# B&R Automation Studio project MotionTestBenchMaster (part 52)

```iecst
                               VAR_DOS_SEQ.Device.LSJ200.ALR := FALSE;                                                 (* STEP: 67 *)
                               VAR_DOS_SEQ.Device.LSJ200.WAIT_OFF := FALSE;
                               VAR_DOS_SEQ.Device.LSJ200.WAIT_ON := FALSE;

                               VAR_DOS_SEQ.Device.LSJ201.ALR := FALSE;                                                 (* STEP: 67 *)
                               VAR_DOS_SEQ.Device.LSJ201.WAIT_OFF := FALSE;
                               VAR_DOS_SEQ.Device.LSJ201.WAIT_ON := FALSE;

                               VAR_DOS_SEQ.Device.LSJ202.ALR := FALSE;                                                 (* STEP: 67 *)
                               VAR_DOS_SEQ.Device.LSJ202.WAIT_OFF := FALSE;
                               VAR_DOS_SEQ.Device.LSJ202.WAIT_ON := FALSE;

                               VAR_DOS_SEQ.Device.FSJ201.ALR := FALSE;                                                 (* STEP: 67 *)
                               VAR_DOS_SEQ.Device.FSJ201.WAIT_OFF := FALSE;
                               VAR_DOS_SEQ.Device.FSJ201.WAIT_ON := FALSE;

                               VAR_DOS_SEQ.Device.FSJ202.ALR := FALSE;                                                 (* STEP: 67 *)
                               VAR_DOS_SEQ.Device.FSJ202.WAIT_OFF := FALSE;
                               VAR_DOS_SEQ.Device.FSJ202.WAIT_ON := FALSE;

                               VAR_DOS_SEQ.Mem.PBAbortEnable := FALSE;                                                 (* STEP: 67 PB Abort Sequence Enable*)
                               VAR_DOS_SEQ.Mem.PBStopEnable := FALSE;                                                  (* STEP: 67 PB Stop Sequence Enable*)
                               VAR_DOS_SEQ.Mem.PBStartEnable := FALSE;                                                 (* STEP: 67 PB Start Sequence Enable*)
                               VAR_DOS_SEQ.Mem.ContainersStop := TRUE;                                                 (* STEP: 67 *)
                               VAR_DOS_SEQ.Mem.MachineStart := TRUE;                                                   (* STEP: 67 *)
                               VAR_DOS_SEQ.Mem.MachineStop := FALSE;                                                   (* STEP: 67 *)
                               VAR_DOS_SEQ.Mem.DummyBottles := FALSE;                                                  (* STEP: 67 Dummy Bottle Install*)
                               VAR_DOS_SEQ.Mem.PositioningRequest := FALSE;                                            (* STEP: 67 Request of Cam Positioning at height SP of Sequncer*)
                               VAR_DOS_SEQ.Mem.COP_Cycle := FALSE;                                                     (* STEP: 67 COP Cycle Check Requested*)
                               VAR_DOS_SEQ.Mem.LapsCounter := FALSE;                                                   (* STEP: 67 *)
                               VAR_DOS_SEQ.Mem.ValveOpening := FALSE;                                                  (* STEP: 67 *)
                               VAR_DOS_SEQ.Mem.CopAfterCipRequest := FALSE;                                            (* STEP: 67 Request Of Cop After Cip*)

                               VAR_DOS_SEQ.ITC.CIP_CleaningRequest := TRUE;                                            (* STEP: 67 To CIP -> Request of Solution Sending*)
                               VAR_DOS_SEQ.ITC.CIP_Alarm := FALSE;                                                     (* STEP: 67 To CIP -> Critical Alarm Present*)
                               VAR_DOS_SEQ.ITC.CIP_RinseEnded := FALSE;                                                (* STEP: 67 To CIP -> Rinse Finished*)
                               VAR_DOS_SEQ.ITC.CIP_ChangeEnded := FALSE;                                               (* STEP: 67 To CIP -> Change Finished*)
                               VAR_DOS_SEQ.ITC.CIP_DrainRunning := FALSE;                                              (* STEP: 67 To CIP -> Drain Cycle Running*)
                               VAR_DOS_SEQ.ITC.CIP_RinseRunning := FALSE;                                              (* STEP: 67 To CIP -> Rinse Cycle Running*)
                               VAR_DOS_SEQ.ITC.CIP_CleaningRunning := TRUE;                                            (* STEP: 67 To CIP -> Cleaning Cycle Running*)
                               VAR_DOS_SEQ.ITC.CIP_DrainEnded := FALSE;                                                (* STEP: 67 To CIP -> Drain Finished*)
                               VAR_DOS_SEQ.ITC.CIP_FloodingEnded := FALSE;                                             (* STEP: 67 To CIP -> Flooding Finished*)
                               VAR_DOS_SEQ.ITC.CIP_FlipEnable := FALSE;                                                (* STEP: 67 *)
                               VAR_DOS_SEQ.ITC.CIP_CycleEnded := FALSE;                                                (* STEP: 67 *)

                               VAR_DOS_SEQ.ITC.PROD_ReadyForHeating := FALSE;                                          (* STEP: 67 To PASTO -> Filler Ready for Production (Heating)*)
                               VAR_DOS_SEQ.ITC.PROD_DoserInTemperature := FALSE;                                       (* STEP: 67 To PASTO -> Filler Temperature OK (After Heating)*)
                               VAR_DOS_SEQ.ITC.PROD_ProductRequest := FALSE;                                           (* STEP: 67 To PASTO -> Product Request*)
                               VAR_DOS_SEQ.ITC.PROD_DoserOnFillingMode := FALSE;                                       (* STEP: 67 To PASTO -> Product Consumend -Filling Valve Opening*)
                               VAR_DOS_SEQ.ITC.PROD_EndProductionCompleted := FALSE;                                   (* STEP: 67 To PASTO -> End Production Done*)
                               VAR_DOS_SEQ.ITC.PROD_ProductRecoveryEnd := FALSE;                                       (* STEP: 67 To PASTO -> Product Recovery End*)
                               VAR_DOS_SEQ.ITC.PROD_WaterRequestAfterProd := FALSE;                                    (* STEP: 67 To PASTO -> Water Request For Filler Rinse Afetr Production*)

                       68: (* CIP - Conical valve extraction 2st group clean *)

                               VAR_DOS_SEQ.Device.PPJ201_PID.PID_Enable := FALSE;                                      (* STEP: 68 Doser Recovery Pump*)
                               VAR_DOS_SEQ.Device.PPJ201_PID.PID_Mode := FALSE;
                               VAR_DOS_SEQ.Device.PPJ201_PID.Auto_SP_Value := 0;
                               VAR_DOS_SEQ.Device.PPJ201_PID.FIX_Value := 0;

                               VAR_DOS_SEQ.Device.PPJ202_PID.PID_Enable := TRUE;                                       (* STEP: 68 Doser Recovery Pump*)
                               VAR_DOS_SEQ.Device.PPJ202_PID.PID_Mode := TRUE;
                               VAR_DOS_SEQ.Device.PPJ202_PID.Auto_SP_Value := 0;
                               VAR_DOS_SEQ.Device.PPJ202_PID.FIX_Value := 15;

                               VAR_DOS_SEQ.Device.PPJ203_PID.PID_Enable := FALSE;                                      (* STEP: 68 Diaphragm Pump for Recovery pulp*)
                               VAR_DOS_SEQ.Device.PPJ203_PID.PID_Mode := FALSE;
                               VAR_DOS_SEQ.Device.PPJ203_PID.Auto_SP_Value := 0;
                               VAR_DOS_SEQ.Device.PPJ203_PID.FIX_Value := 0;

                               VAR_DOS_SEQ.Device.MMJ201_PID.PID_Enable := TRUE;                                       (* STEP: 68 Shaker Motor*)
                               VAR_DOS_SEQ.Device.MMJ201_PID.PID_Mode := TRUE;
                               VAR_DOS_SEQ.Device.MMJ201_PID.Auto_SP_Value := 0;
                               VAR_DOS_SEQ.Device.MMJ201_PID.FIX_Value := 15;

                               VAR_DOS_SEQ.Device.RVJ201_PID.PID_Enable := FALSE;                                      (* STEP: 68 *)
                               VAR_DOS_SEQ.Device.RVJ201_PID.PID_Mode := FALSE;
                               VAR_DOS_SEQ.Device.RVJ201_PID.Auto_SP_Value := 0;
                               VAR_DOS_SEQ.Device.RVJ201_PID.FIX_Value := 0;

                               VAR_DOS_SEQ.Device.AVJ201.AutoCnd := TRUE;                                              (* STEP: 68 Inlet Valve*)
                               VAR_DOS_SEQ.Device.AVJ201.EnableCnd := FALSE;
                               VAR_DOS_SEQ.Device.AVJ210.AutoCnd := FALSE;                                             (* STEP: 68 Washing Duct Valve*)
                               VAR_DOS_SEQ.Device.AVJ210.EnableCnd := FALSE;
                               VAR_DOS_SEQ.Device.AVJ211.AutoCnd := FALSE;                                             (* STEP: 68 Sprayball Valve*)
                               VAR_DOS_SEQ.Device.AVJ211.EnableCnd := FALSE;
                               VAR_DOS_SEQ.Device.AVJ212.AutoCnd := FALSE;                                             (* STEP: 68 *)
                               VAR_DOS_SEQ.Device.AVJ212.EnableCnd := FALSE;
                               VAR_DOS_SEQ.Device.AVJ215.AutoCnd := FALSE;                                             (* STEP: 68 Atmospheric drain valve*)
                               VAR_DOS_SEQ.Device.AVJ215.EnableCnd := FALSE;
                               VAR_DOS_SEQ.Device.AVJ216.AutoCnd := TRUE;                                              (* STEP: 68 Recirculation Valve*)
                               VAR_DOS_SEQ.Device.AVJ216.EnableCnd := FALSE;
                               VAR_DOS_SEQ.Device.AVJ217.AutoCnd := TRUE;                                              (* STEP: 68 Tank Hema Drain Valve*)
                               VAR_DOS_SEQ.Device.AVJ217.EnableCnd := FALSE;
                               VAR_DOS_SEQ.Device.AVJ218.AutoCnd := TRUE;                                              (* STEP: 68 Recirculation Valve*)
                               VAR_DOS_SEQ.Device.AVJ218.EnableCnd := FALSE;
                               VAR_DOS_SEQ.Device.AVJ221.AutoCnd := FALSE;                                             (* STEP: 68 Inlet Loop Valve*)
                               VAR_DOS_SEQ.Device.AVJ221.EnableCnd := FALSE;
                               VAR_DOS_SEQ.Device.AVJ230.AutoCnd := FALSE;                                             (* STEP: 68 *)
                               VAR_DOS_SEQ.Device.AVJ230.EnableCnd := FALSE;
                               VAR_DOS_SEQ.Device.AVJ231.AutoCnd := FALSE;                                             (* STEP: 68 *)
                               VAR_DOS_SEQ.Device.AVJ231.EnableCnd := FALSE;
                               VAR_DOS_SEQ.Device.AVJ232.AutoCnd := FALSE;                                             (* STEP: 68 *)
                               VAR_DOS_SEQ.Device.AVJ232.EnableCnd := FALSE;
                               VAR_DOS_SEQ.Device.AVJ233.AutoCnd := FALSE;                                             (* STEP: 68 *)
                               VAR_DOS_SEQ.Device.AVJ233.EnableCnd := FALSE;
                               VAR_DOS_SEQ.Device.AVJ234.AutoCnd := FALSE;                                             (* STEP: 68 *)
                               VAR_DOS_SEQ.Device.AVJ234.EnableCnd := FALSE;
                               VAR_DOS_SEQ.Device.AVJ235.AutoCnd := FALSE;                                             (* STEP: 68 *)
                               VAR_DOS_SEQ.Device.AVJ235.EnableCnd := FALSE;

                               VAR_DOS_SEQ.Device.LTJ203.ALR_HighLimitEn := FALSE;                                     (* STEP: 68 Hema Tank Level*)
                               VAR_DOS_SEQ.Device.LTJ203.ALR_HighLimitSP := 0;
                               VAR_DOS_SEQ.Device.LTJ203.ALR_LowLimitEn := FALSE;
                               VAR_DOS_SEQ.Device.LTJ203.ALR_LowLimitSP := 0;
                               VAR_DOS_SEQ.Device.LTJ203.SP := 0;
                               VAR_DOS_SEQ.Device.LTJ203.CMP := 0;
                               VAR_DOS_SEQ.Device.LTJ203.MinDev := 0;
                               VAR_DOS_SEQ.Device.LTJ203.MaxDev := 0;

                               VAR_DOS_SEQ.Device.TTJ203.ALR_HighLimitEn := FALSE;                                     (* STEP: 68 Hema Tank Temperature*)
                               VAR_DOS_SEQ.Device.TTJ203.ALR_HighLimitSP := 0;
                               VAR_DOS_SEQ.Device.TTJ203.ALR_LowLimitEn := FALSE;
                               VAR_DOS_SEQ.Device.TTJ203.ALR_LowLimitSP := 0;
                               VAR_DOS_SEQ.Device.TTJ203.SP := 0;
                               VAR_DOS_SEQ.Device.TTJ203.CMP := 0;
                               VAR_DOS_SEQ.Device.TTJ203.MinDev := 0;
                               VAR_DOS_SEQ.Device.TTJ203.MaxDev := 0;

                               VAR_DOS_SEQ.Device.LSJ200.ALR := FALSE;                                                 (* STEP: 68 *)
                               VAR_DOS_SEQ.Device.LSJ200.WAIT_OFF := FALSE;
                               VAR_DOS_SEQ.Device.LSJ200.WAIT_ON := FALSE;

                               VAR_DOS_SEQ.Device.LSJ201.ALR := FALSE;                                                 (* STEP: 68 *)
                               VAR_DOS_SEQ.Device.LSJ201.WAIT_OFF := FALSE;
                               VAR_DOS_SEQ.Device.LSJ201.WAIT_ON := FALSE;

                               VAR_DOS_SEQ.Device.LSJ202.ALR := FALSE;                                                 (* STEP: 68 *)
                               VAR_DOS_SEQ.Device.LSJ202.WAIT_OFF := FALSE;
                               VAR_DOS_SEQ.Device.LSJ202.WAIT_ON := FALSE;

                               VAR_DOS_SEQ.Device.FSJ201.ALR := FALSE;                                                 (* STEP: 68 *)
                               VAR_DOS_SEQ.Device.FSJ201.WAIT_OFF := FALSE;
                               VAR_DOS_SEQ.Device.FSJ201.WAIT_ON := FALSE;

                               VAR_DOS_SEQ.Device.FSJ202.ALR := FALSE;                                                 (* STEP: 68 *)
                               VAR_DOS_SEQ.Device.FSJ202.WAIT_OFF := FALSE;
                               VAR_DOS_SEQ.Device.FSJ202.WAIT_ON := FALSE;

                               VAR_DOS_SEQ.Mem.PBAbortEnable := FALSE;                                                 (* STEP: 68 PB Abort Sequence Enable*)
                               VAR_DOS_SEQ.Mem.PBStopEnable := FALSE;                                                  (* STEP: 68 PB Stop Sequence Enable*)
                               VAR_DOS_SEQ.Mem.PBStartEnable := FALSE;                                                 (* STEP: 68 PB Start Sequence Enable*)
                               VAR_DOS_SEQ.Mem.ContainersStop := TRUE;                                                 (* STEP: 68 *)
                               VAR_DOS_SEQ.Mem.MachineStart := TRUE;                                                   (* STEP: 68 *)
                               VAR_DOS_SEQ.Mem.MachineStop := FALSE;                                                   (* STEP: 68 *)
                               VAR_DOS_SEQ.Mem.DummyBottles := FALSE;                                                  (* STEP: 68 Dummy Bottle Install*)
                               VAR_DOS_SEQ.Mem.PositioningRequest := FALSE;                                            (* STEP: 68 Request of Cam Positioning at height SP of Sequncer*)
                               VAR_DOS_SEQ.Mem.COP_Cycle := FALSE;                                                     (* STEP: 68 COP Cycle Check Requested*)
                               VAR_DOS_SEQ.Mem.LapsCounter := FALSE;                                                   (* STEP: 68 *)
                               VAR_DOS_SEQ.Mem.ValveOpening := FALSE;                                                  (* STEP: 68 *)
                               VAR_DOS_SEQ.Mem.CopAfterCipRequest := FALSE;                                            (* STEP: 68 Request Of Cop After Cip*)

                               VAR_DOS_SEQ.ITC.CIP_CleaningRequest := TRUE;                                            (* STEP: 68 To CIP -> Request of Solution Sending*)
                               VAR_DOS_SEQ.ITC.CIP_Alarm := FALSE;                                                     (* STEP: 68 To CIP -> Critical Alarm Present*)
                               VAR_DOS_SEQ.ITC.CIP_RinseEnded := FALSE;                                                (* STEP: 68 To CIP -> Rinse Finished*)
                               VAR_DOS_SEQ.ITC.CIP_ChangeEnded := FALSE;                                               (* STEP: 68 To CIP -> Change Finished*)
                               VAR_DOS_SEQ.ITC.CIP_DrainRunning := FALSE;                                              (* STEP: 68 To CIP -> Drain Cycle Running*)
                               VAR_DOS_SEQ.ITC.CIP_RinseRunning := FALSE;                                              (* STEP: 68 To CIP -> Rinse Cycle Running*)
                               VAR_DOS_SEQ.ITC.CIP_CleaningRunning := TRUE;                                            (* STEP: 68 To CIP -> Cleaning Cycle Running*)
                               VAR_DOS_SEQ.ITC.CIP_DrainEnded := FALSE;                                                (* STEP: 68 To CIP -> Drain Finished*)
                               VAR_DOS_SEQ.ITC.CIP_FloodingEnded := FALSE;                                             (* STEP: 68 To CIP -> Flooding Finished*)
                               VAR_DOS_SEQ.ITC.CIP_FlipEnable := FALSE;                                                (* STEP: 68 *)
                               VAR_DOS_SEQ.ITC.CIP_CycleEnded := FALSE;                                                (* STEP: 68 *)

                               VAR_DOS_SEQ.ITC.PROD_ReadyForHeating := FALSE;                                          (* STEP: 68 To PASTO -> Filler Ready for Production (Heating)*)
                               VAR_DOS_SEQ.ITC.PROD_DoserInTemperature := FALSE;                                       (* STEP: 68 To PASTO -> Filler Temperature OK (After Heating)*)
                               VAR_DOS_SEQ.ITC.PROD_ProductRequest := FALSE;                                           (* STEP: 68 To PASTO -> Product Request*)
                               VAR_DOS_SEQ.ITC.PROD_DoserOnFillingMode := FALSE;                                       (* STEP: 68 To PASTO -> Product Consumend -Filling Valve Opening*)
                               VAR_DOS_SEQ.ITC.PROD_EndProductionCompleted := FALSE;                                   (* STEP: 68 To PASTO -> End Production Done*)
                               VAR_DOS_SEQ.ITC.PROD_ProductRecoveryEnd := FALSE;                                       (* STEP: 68 To PASTO -> Product Recovery End*)
                               VAR_DOS_SEQ.ITC.PROD_WaterRequestAfterProd := FALSE;                                    (* STEP: 68 To PASTO -> Water Request For Filler Rinse Afetr Production*)

                       69: (* CIP - Conical valve extraction 3st group clean *)

                               VAR_DOS_SEQ.Device.PPJ201_PID.PID_Enable := FALSE;                                      (* STEP: 69 Doser Recovery Pump*)
                               VAR_DOS_SEQ.Device.PPJ201_PID.PID_Mode := FALSE;
                               VAR_DOS_SEQ.Device.PPJ201_PID.Auto_SP_Value := 0;
                               VAR_DOS_SEQ.Device.PPJ201_PID.FIX_Value := 0;

                               VAR_DOS_SEQ.Device.PPJ202_PID.PID_Enable := TRUE;                                       (* STEP: 69 Doser Recovery Pump*)
                               VAR_DOS_SEQ.Device.PPJ202_PID.PID_Mode := TRUE;
                               VAR_DOS_SEQ.Device.PPJ202_PID.Auto_SP_Value := 0;
                               VAR_DOS_SEQ.Device.PPJ202_PID.FIX_Value := 15;

                               VAR_DOS_SEQ.Device.PPJ203_PID.PID_Enable := FALSE;                                      (* STEP: 69 Diaphragm Pump for Recovery pulp*)
                               VAR_DOS_SEQ.Device.PPJ203_PID.PID_Mode := FALSE;
                               VAR_DOS_SEQ.Device.PPJ203_PID.Auto_SP_Value := 0;
                               VAR_DOS_SEQ.Device.PPJ203_PID.FIX_Value := 0;

                               VAR_DOS_SEQ.Device.MMJ201_PID.PID_Enable := TRUE;                                       (* STEP: 69 Shaker Motor*)
                               VAR_DOS_SEQ.Device.MMJ201_PID.PID_Mode := TRUE;
                               VAR_DOS_SEQ.Device.MMJ201_PID.Auto_SP_Value := 0;
                               VAR_DOS_SEQ.Device.MMJ201_PID.FIX_Value := 15;

                               VAR_DOS_SEQ.Device.RVJ201_PID.PID_Enable := FALSE;                                      (* STEP: 69 *)
                               VAR_DOS_SEQ.Device.RVJ201_PID.PID_Mode := FALSE;
                               VAR_DOS_SEQ.Device.RVJ201_PID.Auto_SP_Value := 0;
                               VAR_DOS_SEQ.Device.RVJ201_PID.FIX_Value := 0;

                               VAR_DOS_SEQ.Device.AVJ201.AutoCnd := TRUE;                                              (* STEP: 69 Inlet Valve*)
                               VAR_DOS_SEQ.Device.AVJ201.EnableCnd := FALSE;
                               VAR_DOS_SEQ.Device.AVJ210.AutoCnd := FALSE;                                             (* STEP: 69 Washing Duct Valve*)
                               VAR_DOS_SEQ.Device.AVJ210.EnableCnd := FALSE;
                               VAR_DOS_SEQ.Device.AVJ211.AutoCnd := FALSE;                                             (* STEP: 69 Sprayball Valve*)
                               VAR_DOS_SEQ.Device.AVJ211.EnableCnd := FALSE;
                               VAR_DOS_SEQ.Device.AVJ212.AutoCnd := FALSE;                                             (* STEP: 69 *)
                               VAR_DOS_SEQ.Device.AVJ212.EnableCnd := FALSE;
                               VAR_DOS_SEQ.Device.AVJ215.AutoCnd := FALSE;                                             (* STEP: 69 Atmospheric drain valve*)
                               VAR_DOS_SEQ.Device.AVJ215.EnableCnd := FALSE;
                               VAR_DOS_SEQ.Device.AVJ216.AutoCnd := TRUE;                                              (* STEP: 69 Recirculation Valve*)
                               VAR_DOS_SEQ.Device.AVJ216.EnableCnd := FALSE;
                               VAR_DOS_SEQ.Device.AVJ217.AutoCnd := TRUE;                                              (* STEP: 69 Tank Hema Drain Valve*)
                               VAR_DOS_SEQ.Device.AVJ217.EnableCnd := FALSE;
                               VAR_DOS_SEQ.Device.AVJ218.AutoCnd := TRUE;                                              (* STEP: 69 Recirculation Valve*)
                               VAR_DOS_SEQ.Device.AVJ218.EnableCnd := FALSE;
                               VAR_DOS_SEQ.Device.AVJ221.AutoCnd := FALSE;                                             (* STEP: 69 Inlet Loop Valve*)
                               VAR_DOS_SEQ.Device.AVJ221.EnableCnd := FALSE;
                               VAR_DOS_SEQ.Device.AVJ230.AutoCnd := FALSE;                                             (* STEP: 69 *)
                               VAR_DOS_SEQ.Device.AVJ230.EnableCnd := FALSE;
                               VAR_DOS_SEQ.Device.AVJ231.AutoCnd := FALSE;                                             (* STEP: 69 *)
                               VAR_DOS_SEQ.Device.AVJ231.EnableCnd := FALSE;
                               VAR_DOS_SEQ.Device.AVJ232.AutoCnd := FALSE;                                             (* STEP: 69 *)
                               VAR_DOS_SEQ.Device.AVJ232.EnableCnd := FALSE;
                               VAR_DOS_SEQ.Device.AVJ233.AutoCnd := FALSE;                                             (* STEP: 69 *)
                               VAR_DOS_SEQ.Device.AVJ233.EnableCnd := FALSE;
                               VAR_DOS_SEQ.Device.AVJ234.AutoCnd := FALSE;                                             (* STEP: 69 *)
                               VAR_DOS_SEQ.Device.AVJ234.EnableCnd := FALSE;
                               VAR_DOS_SEQ.Device.AVJ235.AutoCnd := FALSE;                                             (* STEP: 69 *)
                               VAR_DOS_SEQ.Device.AVJ235.EnableCnd := FALSE;

                               VAR_DOS_SEQ.Device.LTJ203.ALR_HighLimitEn := FALSE;                                     (* STEP: 69 Hema Tank Level*)
                               VAR_DOS_SEQ.Device.LTJ203.ALR_HighLimitSP := 0;
                               VAR_DOS_SEQ.Device.LTJ203.ALR_LowLimitEn := FALSE;
                               VAR_DOS_SEQ.Device.LTJ203.ALR_LowLimitSP := 0;
                               VAR_DOS_SEQ.Device.LTJ203.SP := 0;
                               VAR_DOS_SEQ.Device.LTJ203.CMP := 0;
                               VAR_DOS_SEQ.Device.LTJ203.MinDev := 0;
                               VAR_DOS_SEQ.Device.LTJ203.MaxDev := 0;

                               VAR_DOS_SEQ.Device.TTJ203.ALR_HighLimitEn := FALSE;                                     (* STEP: 69 Hema Tank Temperature*)
                               VAR_DOS_SEQ.Device.TTJ203.ALR_HighLimitSP := 0;
                               VAR_DOS_SEQ.Device.TTJ203.ALR_LowLimitEn := FALSE;
                               VAR_DOS_SEQ.Device.TTJ203.ALR_LowLimitSP := 0;
                               VAR_DOS_SEQ.Device.TTJ203.SP := 0;
                               VAR_DOS_SEQ.Device.TTJ203.CMP := 0;
                               VAR_DOS_SEQ.Device.TTJ203.MinDev := 0;
                               VAR_DOS_SEQ.Device.TTJ203.MaxDev := 0;

                               VAR_DOS_SEQ.Device.LSJ200.ALR := FALSE;                                                 (* STEP: 69 *)
                               VAR_DOS_SEQ.Device.LSJ200.WAIT_OFF := FALSE;
                               VAR_DOS_SEQ.Device.LSJ200.WAIT_ON := FALSE;

                               VAR_DOS_SEQ.Device.LSJ201.ALR := FALSE;                                                 (* STEP: 69 *)
                               VAR_DOS_SEQ.Device.LSJ201.WAIT_OFF := FALSE;
                               VAR_DOS_SEQ.Device.LSJ201.WAIT_ON := FALSE;

                               VAR_DOS_SEQ.Device.LSJ202.ALR := FALSE;                                                 (* STEP: 69 *)
                               VAR_DOS_SEQ.Device.LSJ202.WAIT_OFF := FALSE;
                               VAR_DOS_SEQ.Device.LSJ202.WAIT_ON := FALSE;

                               VAR_DOS_SEQ.Device.FSJ201.ALR := FALSE;                                                 (* STEP: 69 *)
                               VAR_DOS_SEQ.Device.FSJ201.WAIT_OFF := FALSE;
                               VAR_DOS_SEQ.Device.FSJ201.WAIT_ON := FALSE;

                               VAR_DOS_SEQ.Device.FSJ202.ALR := FALSE;                                                 (* STEP: 69 *)
                               VAR_DOS_SEQ.Device.FSJ202.WAIT_OFF := FALSE;
                               VAR_DOS_SEQ.Device.FSJ202.WAIT_ON := FALSE;

                               VAR_DOS_SEQ.Mem.PBAbortEnable := FALSE;                                                 (* STEP: 69 PB Abort Sequence Enable*)
                               VAR_DOS_SEQ.Mem.PBStopEnable := FALSE;                                                  (* STEP: 69 PB Stop Sequence Enable*)
                               VAR_DOS_SEQ.Mem.PBStartEnable := FALSE;                                                 (* STEP: 69 PB Start Sequence Enable*)
                               VAR_DOS_SEQ.Mem.ContainersStop := TRUE;                                                 (* STEP: 69 *)
                               VAR_DOS_SEQ.Mem.MachineStart := TRUE;                                                   (* STEP: 69 *)
                               VAR_DOS_SEQ.Mem.MachineStop := FALSE;                                                   (* STEP: 69 *)
                               VAR_DOS_SEQ.Mem.DummyBottles := FALSE;                                                  (* STEP: 69 Dummy Bottle Install*)
                               VAR_DOS_SEQ.Mem.PositioningRequest := FALSE;                                            (* STEP: 69 Request of Cam Positioning at height SP of Sequncer*)
                               VAR_DOS_SEQ.Mem.COP_Cycle := FALSE;                                                     (* STEP: 69 COP Cycle Check Requested*)
                               VAR_DOS_SEQ.Mem.LapsCounter := FALSE;                                                   (* STEP: 69 *)
                               VAR_DOS_SEQ.Mem.ValveOpening := FALSE;                                                  (* STEP: 69 *)
                               VAR_DOS_SEQ.Mem.CopAfterCipRequest := FALSE;                                            (* STEP: 69 Request Of Cop After Cip*)

                               VAR_DOS_SEQ.ITC.CIP_CleaningRequest := TRUE;                                            (* STEP: 69 To CIP -> Request of Solution Sending*)
                               VAR_DOS_SEQ.ITC.CIP_Alarm := FALSE;                                                     (* STEP: 69 To CIP -> Critical Alarm Present*)
                               VAR_DOS_SEQ.ITC.CIP_RinseEnded := FALSE;                                                (* STEP: 69 To CIP -> Rinse Finished*)
                               VAR_DOS_SEQ.ITC.CIP_ChangeEnded := FALSE;                                               (* STEP: 69 To CIP -> Change Finished*)
                               VAR_DOS_SEQ.ITC.CIP_DrainRunning := FALSE;                                              (* STEP: 69 To CIP -> Drain Cycle Running*)
                               VAR_DOS_SEQ.ITC.CIP_RinseRunning := FALSE;                                              (* STEP: 69 To CIP -> Rinse Cycle Running*)
                               VAR_DOS_SEQ.ITC.CIP_CleaningRunning := TRUE;                                            (* STEP: 69 To CIP -> Cleaning Cycle Running*)
                               VAR_DOS_SEQ.ITC.CIP_DrainEnded := FALSE;                                                (* STEP: 69 To CIP -> Drain Finished*)
                               VAR_DOS_SEQ.ITC.CIP_FloodingEnded := FALSE;                                             (* STEP: 69 To CIP -> Flooding Finished*)
                               VAR_DOS_SEQ.ITC.CIP_FlipEnable := FALSE;                                                (* STEP: 69 *)
                               VAR_DOS_SEQ.ITC.CIP_CycleEnded := FALSE;                                                (* STEP: 69 *)

                               VAR_DOS_SEQ.ITC.PROD_ReadyForHeating := FALSE;                                          (* STEP: 69 To PASTO -> Filler Ready for Production (Heating)*)
                               VAR_DOS_SEQ.ITC.PROD_DoserInTemperature := FALSE;                                       (* STEP: 69 To PASTO -> Filler Temperature OK (After Heating)*)
                               VAR_DOS_SEQ.ITC.PROD_ProductRequest := FALSE;                                           (* STEP: 69 To PASTO -> Product Request*)
                               VAR_DOS_SEQ.ITC.PROD_DoserOnFillingMode := FALSE;                                       (* STEP: 69 To PASTO -> Product Consumend -Filling Valve Opening*)
                               VAR_DOS_SEQ.ITC.PROD_EndProductionCompleted := FALSE;                                   (* STEP: 69 To PASTO -> End Production Done*)
                               VAR_DOS_SEQ.ITC.PROD_ProductRecoveryEnd := FALSE;                                       (* STEP: 69 To PASTO -> Product Recovery End*)
                               VAR_DOS_SEQ.ITC.PROD_WaterRequestAfterProd := FALSE;                                    (* STEP: 69 To PASTO -> Water Request For Filler Rinse Afetr Production*)

                       70: (* CIP - Conical valve exctraction drain *)

                               VAR_DOS_SEQ.Device.PPJ201_PID.PID_Enable := FALSE;                                      (* STEP: 70 Doser Recovery Pump*)
                               VAR_DOS_SEQ.Device.PPJ201_PID.PID_Mode := FALSE;
                               VAR_DOS_SEQ.Device.PPJ201_PID.Auto_SP_Value := 0;
                               VAR_DOS_SEQ.Device.PPJ201_PID.FIX_Value := 0;

                               VAR_DOS_SEQ.Device.PPJ202_PID.PID_Enable := TRUE;                                       (* STEP: 70 Doser Recovery Pump*)
                               VAR_DOS_SEQ.Device.PPJ202_PID.PID_Mode := FALSE;
                               VAR_DOS_SEQ.Device.PPJ202_PID.Auto_SP_Value := 0;
                               VAR_DOS_SEQ.Device.PPJ202_PID.FIX_Value := 15;

                               VAR_DOS_SEQ.Device.PPJ203_PID.PID_Enable := FALSE;                                      (* STEP: 70 Diaphragm Pump for Recovery pulp*)
                               VAR_DOS_SEQ.Device.PPJ203_PID.PID_Mode := FALSE;
                               VAR_DOS_SEQ.Device.PPJ203_PID.Auto_SP_Value := 0;
                               VAR_DOS_SEQ.Device.PPJ203_PID.FIX_Value := 0;

                               VAR_DOS_SEQ.Device.MMJ201_PID.PID_Enable := FALSE;                                      (* STEP: 70 Shaker Motor*)
                               VAR_DOS_SEQ.Device.MMJ201_PID.PID_Mode := FALSE;
                               VAR_DOS_SEQ.Device.MMJ201_PID.Auto_SP_Value := 0;
                               VAR_DOS_SEQ.Device.MMJ201_PID.FIX_Value := 0;

                               VAR_DOS_SEQ.Device.RVJ201_PID.PID_Enable := FALSE;                                      (* STEP: 70 *)
                               VAR_DOS_SEQ.Device.RVJ201_PID.PID_Mode := FALSE;
                               VAR_DOS_SEQ.Device.RVJ201_PID.Auto_SP_Value := 0;
                               VAR_DOS_SEQ.Device.RVJ201_PID.FIX_Value := 0;

                               VAR_DOS_SEQ.Device.AVJ201.AutoCnd := FALSE;                                             (* STEP: 70 Inlet Valve*)
                               VAR_DOS_SEQ.Device.AVJ201.EnableCnd := FALSE;
                               VAR_DOS_SEQ.Device.AVJ210.AutoCnd := FALSE;                                             (* STEP: 70 Washing Duct Valve*)
                               VAR_DOS_SEQ.Device.AVJ210.EnableCnd := FALSE;
                               VAR_DOS_SEQ.Device.AVJ211.AutoCnd := FALSE;                                             (* STEP: 70 Sprayball Valve*)
                               VAR_DOS_SEQ.Device.AVJ211.EnableCnd := FALSE;
                               VAR_DOS_SEQ.Device.AVJ212.AutoCnd := FALSE;                                             (* STEP: 70 *)
                               VAR_DOS_SEQ.Device.AVJ212.EnableCnd := FALSE;
                               VAR_DOS_SEQ.Device.AVJ215.AutoCnd := FALSE;                                             (* STEP: 70 Atmospheric drain valve*)
                               VAR_DOS_SEQ.Device.AVJ215.EnableCnd := FALSE;
                               VAR_DOS_SEQ.Device.AVJ216.AutoCnd := TRUE;                                              (* STEP: 70 Recirculation Valve*)
                               VAR_DOS_SEQ.Device.AVJ216.EnableCnd := FALSE;
                               VAR_DOS_SEQ.Device.AVJ217.AutoCnd := TRUE;                                              (* STEP: 70 Tank Hema Drain Valve*)
                               VAR_DOS_SEQ.Device.AVJ217.EnableCnd := FALSE;
                               VAR_DOS_SEQ.Device.AVJ218.AutoCnd := TRUE;                                              (* STEP: 70 Recirculation Valve*)
                               VAR_DOS_SEQ.Device.AVJ218.EnableCnd := FALSE;
                               VAR_DOS_SEQ.Device.AVJ221.AutoCnd := FALSE;                                             (* STEP: 70 Inlet Loop Valve*)
                               VAR_DOS_SEQ.Device.AVJ221.EnableCnd := FALSE;
                               VAR_DOS_SEQ.Device.AVJ230.AutoCnd := FALSE;                                             (* STEP: 70 *)
                               VAR_DOS_SEQ.Device.AVJ230.EnableCnd := FALSE;
                               VAR_DOS_SEQ.Device.AVJ231.AutoCnd := FALSE;                                             (* STEP: 70 *)
                               VAR_DOS_SEQ.Device.AVJ231.EnableCnd := FALSE;
                               VAR_DOS_SEQ.Device.AVJ232.AutoCnd := FALSE;                                             (* STEP: 70 *)
                               VAR_DOS_SEQ.Device.AVJ232.EnableCnd := FALSE;
                               VAR_DOS_SEQ.Device.AVJ233.AutoCnd := FALSE;                                             (* STEP: 70 *)
                               VAR_DOS_SEQ.Device.AVJ233.EnableCnd := FALSE;
                               VAR_DOS_SEQ.Device.AVJ234.AutoCnd := FALSE;                                             (* STEP: 70 *)
                               VAR_DOS_SEQ.Device.AVJ234.EnableCnd := FALSE;
                               VAR_DOS_SEQ.Device.AVJ235.AutoCnd := FALSE;                                             (* STEP: 70 *)
                               VAR_DOS_SEQ.Device.AVJ235.EnableCnd := FALSE;

                               VAR_DOS_SEQ.Device.LTJ203.ALR_HighLimitEn := FALSE;                                     (* STEP: 70 Hema Tank Level*)
                               VAR_DOS_SEQ.Device.LTJ203.ALR_HighLimitSP := 0;
                               VAR_DOS_SEQ.Device.LTJ203.ALR_LowLimitEn := FALSE;
                               VAR_DOS_SEQ.Device.LTJ203.ALR_LowLimitSP := 0;
                               VAR_DOS_SEQ.Device.LTJ203.SP := 0;
                               VAR_DOS_SEQ.Device.LTJ203.CMP := 0;
                               VAR_DOS_SEQ.Device.LTJ203.MinDev := 0;
                               VAR_DOS_SEQ.Device.LTJ203.MaxDev := 0;

                               VAR_DOS_SEQ.Device.TTJ203.ALR_HighLimitEn := FALSE;                                     (* STEP: 70 Hema Tank Temperature*)
                               VAR_DOS_SEQ.Device.TTJ203.ALR_HighLimitSP := 0;
                               VAR_DOS_SEQ.Device.TTJ203.ALR_LowLimitEn := FALSE;
                               VAR_DOS_SEQ.Device.TTJ203.ALR_LowLimitSP := 0;
                               VAR_DOS_SEQ.Device.TTJ203.SP := 0;
                               VAR_DOS_SEQ.Device.TTJ203.CMP := 0;
                               VAR_DOS_SEQ.Device.TTJ203.MinDev := 0;
                               VAR_DOS_SEQ.Device.TTJ203.MaxDev := 0;

                               VAR_DOS_SEQ.Device.LSJ200.ALR := FALSE;                                                 (* STEP: 70 *)
                               VAR_DOS_SEQ.Device.LSJ200.WAIT_OFF := FALSE;
                               VAR_DOS_SEQ.Device.LSJ200.WAIT_ON := FALSE;

                               VAR_DOS_SEQ.Device.LSJ201.ALR := FALSE;                                                 (* STEP: 70 *)
                               VAR_DOS_SEQ.Device.LSJ201.WAIT_OFF := FALSE;
                               VAR_DOS_SEQ.Device.LSJ201.WAIT_ON := FALSE;

                               VAR_DOS_SEQ.Device.LSJ202.ALR := FALSE;                                                 (* STEP: 70 *)
                               VAR_DOS_SEQ.Device.LSJ202.WAIT_OFF := FALSE;
                               VAR_DOS_SEQ.Device.LSJ202.WAIT_ON := FALSE;

                               VAR_DOS_SEQ.Device.FSJ201.ALR := FALSE;                                                 (* STEP: 70 *)
                               VAR_DOS_SEQ.Device.FSJ201.WAIT_OFF := FALSE;
                               VAR_DOS_SEQ.Device.FSJ201.WAIT_ON := FALSE;

                               VAR_DOS_SEQ.Device.FSJ202.ALR := FALSE;                                                 (* STEP: 70 *)
                               VAR_DOS_SEQ.Device.FSJ202.WAIT_OFF := FALSE;
                               VAR_DOS_SEQ.Device.FSJ202.WAIT_ON := FALSE;

                               VAR_DOS_SEQ.Mem.PBAbortEnable := FALSE;                                                 (* STEP: 70 PB Abort Sequence Enable*)
                               VAR_DOS_SEQ.Mem.PBStopEnable := FALSE;                                                  (* STEP: 70 PB Stop Sequence Enable*)
                               VAR_DOS_SEQ.Mem.PBStartEnable := FALSE;                                                 (* STEP: 70 PB Start Sequence Enable*)
                               VAR_DOS_SEQ.Mem.ContainersStop := TRUE;                                                 (* STEP: 70 *)
                               VAR_DOS_SEQ.Mem.MachineStart := TRUE;                                                   (* STEP: 70 *)
                               VAR_DOS_SEQ.Mem.MachineStop := FALSE;                                                   (* STEP: 70 *)
                               VAR_DOS_SEQ.Mem.DummyBottles := FALSE;                                                  (* STEP: 70 Dummy Bottle Install*)
                               VAR_DOS_SEQ.Mem.PositioningRequest := FALSE;                                            (* STEP: 70 Request of Cam Positioning at height SP of Sequncer*)
                               VAR_DOS_SEQ.Mem.COP_Cycle := FALSE;                                                     (* STEP: 70 COP Cycle Check Requested*)
                               VAR_DOS_SEQ.Mem.LapsCounter := FALSE;                                                   (* STEP: 70 *)
                               VAR_DOS_SEQ.Mem.ValveOpening := FALSE;                                                  (* STEP: 70 *)
                               VAR_DOS_SEQ.Mem.CopAfterCipRequest := FALSE;                                            (* STEP: 70 Request Of Cop After Cip*)

                               VAR_DOS_SEQ.ITC.CIP_CleaningRequest := TRUE;                                            (* STEP: 70 To CIP -> Request of Solution Sending*)
                               VAR_DOS_SEQ.ITC.CIP_Alarm := FALSE;                                                     (* STEP: 70 To CIP -> Critical Alarm Present*)
                               VAR_DOS_SEQ.ITC.CIP_RinseEnded := FALSE;                                                (* STEP: 70 To CIP -> Rinse Finished*)
                               VAR_DOS_SEQ.ITC.CIP_ChangeEnded := FALSE;                                               (* STEP: 70 To CIP -> Change Finished*)
                               VAR_DOS_SEQ.ITC.CIP_DrainRunning := FALSE;                                              (* STEP: 70 To CIP -> Drain Cycle Running*)
                               VAR_DOS_SEQ.ITC.CIP_RinseRunning := FALSE;                                              (* STEP: 70 To CIP -> Rinse Cycle Running*)
                               VAR_DOS_SEQ.ITC.CIP_CleaningRunning := TRUE;                                            (* STEP: 70 To CIP -> Cleaning Cycle Running*)
                               VAR_DOS_SEQ.ITC.CIP_DrainEnded := FALSE;                                                (* STEP: 70 To CIP -> Drain Finished*)
                               VAR_DOS_SEQ.ITC.CIP_FloodingEnded := FALSE;                                             (* STEP: 70 To CIP -> Flooding Finished*)
                               VAR_DOS_SEQ.ITC.CIP_FlipEnable := FALSE;                                                (* STEP: 70 *)
                               VAR_DOS_SEQ.ITC.CIP_CycleEnded := FALSE;                                                (* STEP: 70 *)

                               VAR_DOS_SEQ.ITC.PROD_ReadyForHeating := FALSE;                                          (* STEP: 70 To PASTO -> Filler Ready for Production (Heating)*)
                               VAR_DOS_SEQ.ITC.PROD_DoserInTemperature := FALSE;                                       (* STEP: 70 To PASTO -> Filler Temperature OK (After Heating)*)
                               VAR_DOS_SEQ.ITC.PROD_ProductRequest := FALSE;                                           (* STEP: 70 To PASTO -> Product Request*)
                               VAR_DOS_SEQ.ITC.PROD_DoserOnFillingMode := FALSE;                                       (* STEP: 70 To PASTO -> Product Consumend -Filling Valve Opening*)
                               VAR_DOS_SEQ.ITC.PROD_EndProductionCompleted := FALSE;                                   (* STEP: 70 To PASTO -> End Production Done*)
                               VAR_DOS_SEQ.ITC.PROD_ProductRecoveryEnd := FALSE;                                       (* STEP: 70 To PASTO -> Product Recovery End*)
                               VAR_DOS_SEQ.ITC.PROD_WaterRequestAfterProd := FALSE;                                    (* STEP: 70 To PASTO -> Water Request For Filler Rinse Afetr Production*)

                       71: (* CIP - Conical valve insertion *)

                               VAR_DOS_SEQ.Device.PPJ201_PID.PID_Enable := FALSE;                                      (* STEP: 71 Doser Recovery Pump*)
                               VAR_DOS_SEQ.Device.PPJ201_PID.PID_Mode := FALSE;
                               VAR_DOS_SEQ.Device.PPJ201_PID.Auto_SP_Value := 0;
                               VAR_DOS_SEQ.Device.PPJ201_PID.FIX_Value := 0;

                               VAR_DOS_SEQ.Device.PPJ202_PID.PID_Enable := TRUE;                                       (* STEP: 71 Doser Recovery Pump*)
                               VAR_DOS_SEQ.Device.PPJ202_PID.PID_Mode := FALSE;
                               VAR_DOS_SEQ.Device.PPJ202_PID.Auto_SP_Value := 0;
                               VAR_DOS_SEQ.Device.PPJ202_PID.FIX_Value := 15;

                               VAR_DOS_SEQ.Device.PPJ203_PID.PID_Enable := FALSE;                                      (* STEP: 71 Diaphragm Pump for Recovery pulp*)
                               VAR_DOS_SEQ.Device.PPJ203_PID.PID_Mode := FALSE;
                               VAR_DOS_SEQ.Device.PPJ203_PID.Auto_SP_Value := 0;
                               VAR_DOS_SEQ.Device.PPJ203_PID.FIX_Value := 0;

                               VAR_DOS_SEQ.Device.MMJ201_PID.PID_Enable := FALSE;                                      (* STEP: 71 Shaker Motor*)
                               VAR_DOS_SEQ.Device.MMJ201_PID.PID_Mode := FALSE;
                               VAR_DOS_SEQ.Device.MMJ201_PID.Auto_SP_Value := 0;
                               VAR_DOS_SEQ.Device.MMJ201_PID.FIX_Value := 0;

                               VAR_DOS_SEQ.Device.RVJ201_PID.PID_Enable := FALSE;                                      (* STEP: 71 *)
                               VAR_DOS_SEQ.Device.RVJ201_PID.PID_Mode := FALSE;
                               VAR_DOS_SEQ.Device.RVJ201_PID.Auto_SP_Value := 0;
                               VAR_DOS_SEQ.Device.RVJ201_PID.FIX_Value := 0;

                               VAR_DOS_SEQ.Device.AVJ201.AutoCnd := FALSE;                                             (* STEP: 71 Inlet Valve*)
                               VAR_DOS_SEQ.Device.AVJ201.EnableCnd := FALSE;
                               VAR_DOS_SEQ.Device.AVJ210.AutoCnd := FALSE;                                             (* STEP: 71 Washing Duct Valve*)
                               VAR_DOS_SEQ.Device.AVJ210.EnableCnd := FALSE;
                               VAR_DOS_SEQ.Device.AVJ211.AutoCnd := FALSE;                                             (* STEP: 71 Sprayball Valve*)
                               VAR_DOS_SEQ.Device.AVJ211.EnableCnd := FALSE;
                               VAR_DOS_SEQ.Device.AVJ212.AutoCnd := FALSE;                                             (* STEP: 71 *)
                               VAR_DOS_SEQ.Device.AVJ212.EnableCnd := FALSE;
                               VAR_DOS_SEQ.Device.AVJ215.AutoCnd := FALSE;                                             (* STEP: 71 Atmospheric drain valve*)
                               VAR_DOS_SEQ.Device.AVJ215.EnableCnd := FALSE;
                               VAR_DOS_SEQ.Device.AVJ216.AutoCnd := TRUE;                                              (* STEP: 71 Recirculation Valve*)
                               VAR_DOS_SEQ.Device.AVJ216.EnableCnd := FALSE;
                               VAR_DOS_SEQ.Device.AVJ217.AutoCnd := TRUE;                                              (* STEP: 71 Tank Hema Drain Valve*)
                               VAR_DOS_SEQ.Device.AVJ217.EnableCnd := FALSE;
                               VAR_DOS_SEQ.Device.AVJ218.AutoCnd := TRUE;                                              (* STEP: 71 Recirculation Valve*)
                               VAR_DOS_SEQ.Device.AVJ218.EnableCnd := FALSE;
                               VAR_DOS_SEQ.Device.AVJ221.AutoCnd := FALSE;                                             (* STEP: 71 Inlet Loop Valve*)
                               VAR_DOS_SEQ.Device.AVJ221.EnableCnd := FALSE;
                               VAR_DOS_SEQ.Device.AVJ230.AutoCnd := FALSE;                                             (* STEP: 71 *)
                               VAR_DOS_SEQ.Device.AVJ230.EnableCnd := FALSE;
                               VAR_DOS_SEQ.Device.AVJ231.AutoCnd := FALSE;                                             (* STEP: 71 *)
                               VAR_DOS_SEQ.Device.AVJ231.EnableCnd := FALSE;
                               VAR_DOS_SEQ.Device.AVJ232.AutoCnd := FALSE;                                             (* STEP: 71 *)
                               VAR_DOS_SEQ.Device.AVJ232.EnableCnd := FALSE;
                               VAR_DOS_SEQ.Device.AVJ233.AutoCnd := FALSE;                                             (* STEP: 71 *)
                               VAR_DOS_SEQ.Device.AVJ233.EnableCnd := FALSE;
                               VAR_DOS_SEQ.Device.AVJ234.AutoCnd := FALSE;                                             (* STEP: 71 *)
                               VAR_DOS_SEQ.Device.AVJ234.EnableCnd := FALSE;
                               VAR_DOS_SEQ.Device.AVJ235.AutoCnd := FALSE;                                             (* STEP: 71 *)
                               VAR_DOS_SEQ.Device.AVJ235.EnableCnd := FALSE;

                               VAR_DOS_SEQ.Device.LTJ203.ALR_HighLimitEn := FALSE;                                     (* STEP: 71 Hema Tank Level*)
                               VAR_DOS_SEQ.Device.LTJ203.ALR_HighLimitSP := 0;
                               VAR_DOS_SEQ.Device.LTJ203.ALR_LowLimitEn := FALSE;
                               VAR_DOS_SEQ.Device.LTJ203.ALR_LowLimitSP := 0;
                               VAR_DOS_SEQ.Device.LTJ203.SP := 0;
                               VAR_DOS_SEQ.Device.LTJ203.CMP := 0;
                               VAR_DOS_SEQ.Device.LTJ203.MinDev := 0;
                               VAR_DOS_SEQ.Device.LTJ203.MaxDev := 0;

                               VAR_DOS_SEQ.Device.TTJ203.ALR_HighLimitEn := FALSE;                                     (* STEP: 71 Hema Tank Temperature*)
                               VAR_DOS_SEQ.Device.TTJ203.ALR_HighLimitSP := 0;
                               VAR_DOS_SEQ.Device.TTJ203.ALR_LowLimitEn := FALSE;
                               VAR_DOS_SEQ.Device.TTJ203.ALR_LowLimitSP := 0;
                               VAR_DOS_SEQ.Device.TTJ203.SP := 0;
                               VAR_DOS_SEQ.Device.TTJ203.CMP := 0;
                               VAR_DOS_SEQ.Device.TTJ203.MinDev := 0;
                               VAR_DOS_SEQ.Device.TTJ203.MaxDev := 0;

                               VAR_DOS_SEQ.Device.LSJ200.ALR := FALSE;                                                 (* STEP: 71 *)
                               VAR_DOS_SEQ.Device.LSJ200.WAIT_OFF := FALSE;
                               VAR_DOS_SEQ.Device.LSJ200.WAIT_ON := FALSE;

                               VAR_DOS_SEQ.Device.LSJ201.ALR := FALSE;                                                 (* STEP: 71 *)
                               VAR_DOS_SEQ.Device.LSJ201.WAIT_OFF := FALSE;
                               VAR_DOS_SEQ.Device.LSJ201.WAIT_ON := FALSE;

                               VAR_DOS_SEQ.Device.LSJ202.ALR := FALSE;                                                 (* STEP: 71 *)
                               VAR_DOS_SEQ.Device.LSJ202.WAIT_OFF := FALSE;
                               VAR_DOS_SEQ.Device.LSJ202.WAIT_ON := FALSE;

                               VAR_DOS_SEQ.Device.FSJ201.ALR := FALSE;                                                 (* STEP: 71 *)
                               VAR_DOS_SEQ.Device.FSJ201.WAIT_OFF := FALSE;
                               VAR_DOS_SEQ.Device.FSJ201.WAIT_ON := FALSE;

                               VAR_DOS_SEQ.Device.FSJ202.ALR := FALSE;                                                 (* STEP: 71 *)
                               VAR_DOS_SEQ.Device.FSJ202.WAIT_OFF := FALSE;
                               VAR_DOS_SEQ.Device.FSJ202.WAIT_ON := FALSE;

                               VAR_DOS_SEQ.Mem.PBAbortEnable := FALSE;                                                 (* STEP: 71 PB Abort Sequence Enable*)
                               VAR_DOS_SEQ.Mem.PBStopEnable := FALSE;                                                  (* STEP: 71 PB Stop Sequence Enable*)
                               VAR_DOS_SEQ.Mem.PBStartEnable := FALSE;                                                 (* STEP: 71 PB Start Sequence Enable*)
                               VAR_DOS_SEQ.Mem.ContainersStop := TRUE;                                                 (* STEP: 71 *)
                               VAR_DOS_SEQ.Mem.MachineStart := TRUE;                                                   (* STEP: 71 *)
                               VAR_DOS_SEQ.Mem.MachineStop := FALSE;                                                   (* STEP: 71 *)
                               VAR_DOS_SEQ.Mem.DummyBottles := FALSE;                                                  (* STEP: 71 Dummy Bottle Install*)
                               VAR_DOS_SEQ.Mem.PositioningRequest := FALSE;                                            (* STEP: 71 Request of Cam Positioning at height SP of Sequncer*)
                               VAR_DOS_SEQ.Mem.COP_Cycle := FALSE;                                                     (* STEP: 71 COP Cycle Check Requested*)
                               VAR_DOS_SEQ.Mem.LapsCounter := FALSE;                                                   (* STEP: 71 *)
                               VAR_DOS_SEQ.Mem.ValveOpening := FALSE;                                                  (* STEP: 71 *)
                               VAR_DOS_SEQ.Mem.CopAfterCipRequest := FALSE;                                            (* STEP: 71 Request Of Cop After Cip*)

                               VAR_DOS_SEQ.ITC.CIP_CleaningRequest := TRUE;                                            (* STEP: 71 To CIP -> Request of Solution Sending*)
                               VAR_DOS_SEQ.ITC.CIP_Alarm := FALSE;                                                     (* STEP: 71 To CIP -> Critical Alarm Present*)
                               VAR_DOS_SEQ.ITC.CIP_RinseEnded := FALSE;                                                (* STEP: 71 To CIP -> Rinse Finished*)
                               VAR_DOS_SEQ.ITC.CIP_ChangeEnded := FALSE;                                               (* STEP: 71 To CIP -> Change Finished*)
                               VAR_DOS_SEQ.ITC.CIP_DrainRunning := FALSE;                                              (* STEP: 71 To CIP -> Drain Cycle Running*)
                               VAR_DOS_SEQ.ITC.CIP_RinseRunning := FALSE;                                              (* STEP: 71 To CIP -> Rinse Cycle Running*)
                               VAR_DOS_SEQ.ITC.CIP_CleaningRunning := TRUE;                                            (* STEP: 71 To CIP -> Cleaning Cycle Running*)
                               VAR_DOS_SEQ.ITC.CIP_DrainEnded := FALSE;                                                (* STEP: 71 To CIP -> Drain Finished*)
                               VAR_DOS_SEQ.ITC.CIP_FloodingEnded := FALSE;                                             (* STEP: 71 To CIP -> Flooding Finished*)
                               VAR_DOS_SEQ.ITC.CIP_FlipEnable := FALSE;                                                (* STEP: 71 *)
                               VAR_DOS_SEQ.ITC.CIP_CycleEnded := FALSE;                                                (* STEP: 71 *)

                               VAR_DOS_SEQ.ITC.PROD_ReadyForHeating := FALSE;                                          (* STEP: 71 To PASTO -> Filler Ready for Production (Heating)*)
                               VAR_DOS_SEQ.ITC.PROD_DoserInTemperature := FALSE;                                       (* STEP: 71 To PASTO -> Filler Temperature OK (After Heating)*)
                               VAR_DOS_SEQ.ITC.PROD_ProductRequest := FALSE;                                           (* STEP: 71 To PASTO -> Product Request*)
                               VAR_DOS_SEQ.ITC.PROD_DoserOnFillingMode := FALSE;                                       (* STEP: 71 To PASTO -> Product Consumend -Filling Valve Opening*)
                               VAR_DOS_SEQ.ITC.PROD_EndProductionCompleted := FALSE;                                   (* STEP: 71 To PASTO -> End Production Done*)
                               VAR_DOS_SEQ.ITC.PROD_ProductRecoveryEnd := FALSE;                                       (* STEP: 71 To PASTO -> Product Recovery End*)
                               VAR_DOS_SEQ.ITC.PROD_WaterRequestAfterProd := FALSE;                                    (* STEP: 71 To PASTO -> Water Request For Filler Rinse Afetr Production*)

                       72: (* Spare Steps *)

                       73: (* CIP - Wait for product tank at CIP level *)

                               VAR_DOS_SEQ.Device.PPJ201_PID.PID_Enable := FALSE;                                      (* STEP: 73 Doser Recovery Pump*)
                               VAR_DOS_SEQ.Device.PPJ201_PID.PID_Mode := FALSE;
                               VAR_DOS_SEQ.Device.PPJ201_PID.Auto_SP_Value := 0;
                               VAR_DOS_SEQ.Device.PPJ201_PID.FIX_Value := 0;

                               VAR_DOS_SEQ.Device.PPJ202_PID.PID_Enable := FALSE;                                      (* STEP: 73 Doser Recovery Pump*)
                               VAR_DOS_SEQ.Device.PPJ202_PID.PID_Mode := FALSE;
                               VAR_DOS_SEQ.Device.PPJ202_PID.Auto_SP_Value := 0;
                               VAR_DOS_SEQ.Device.PPJ202_PID.FIX_Value := 0;

                               VAR_DOS_SEQ.Device.PPJ203_PID.PID_Enable := FALSE;                                      (* STEP: 73 Diaphragm Pump for Recovery pulp*)
                               VAR_DOS_SEQ.Device.PPJ203_PID.PID_Mode := FALSE;
                               VAR_DOS_SEQ.Device.PPJ203_PID.Auto_SP_Value := 0;
                               VAR_DOS_SEQ.Device.PPJ203_PID.FIX_Value := 0;

                               VAR_DOS_SEQ.Device.MMJ201_PID.PID_Enable := FALSE;                                      (* STEP: 73 Shaker Motor*)
                               VAR_DOS_SEQ.Device.MMJ201_PID.PID_Mode := FALSE;
                               VAR_DOS_SEQ.Device.MMJ201_PID.Auto_SP_Value := 0;
                               VAR_DOS_SEQ.Device.MMJ201_PID.FIX_Value := 0;

                               VAR_DOS_SEQ.Device.RVJ201_PID.PID_Enable := FALSE;                                      (* STEP: 73 *)
                               VAR_DOS_SEQ.Device.RVJ201_PID.PID_Mode := FALSE;
                               VAR_DOS_SEQ.Device.RVJ201_PID.Auto_SP_Value := 0;
                               VAR_DOS_SEQ.Device.RVJ201_PID.FIX_Value := 0;

                               VAR_DOS_SEQ.Device.AVJ201.AutoCnd := TRUE;                                              (* STEP: 73 Inlet Valve*)
                               VAR_DOS_SEQ.Device.AVJ201.EnableCnd := TRUE;
                               VAR_DOS_SEQ.Device.AVJ210.AutoCnd := FALSE;                                             (* STEP: 73 Washing Duct Valve*)
                               VAR_DOS_SEQ.Device.AVJ210.EnableCnd := FALSE;
                               VAR_DOS_SEQ.Device.AVJ211.AutoCnd := FALSE;                                             (* STEP: 73 Sprayball Valve*)
                               VAR_DOS_SEQ.Device.AVJ211.EnableCnd := FALSE;
                               VAR_DOS_SEQ.Device.AVJ212.AutoCnd := FALSE;                                             (* STEP: 73 *)
                               VAR_DOS_SEQ.Device.AVJ212.EnableCnd := FALSE;
                               VAR_DOS_SEQ.Device.AVJ215.AutoCnd := FALSE;                                             (* STEP: 73 Atmospheric drain valve*)
                               VAR_DOS_SEQ.Device.AVJ215.EnableCnd := FALSE;
                               VAR_DOS_SEQ.Device.AVJ216.AutoCnd := TRUE;                                              (* STEP: 73 Recirculation Valve*)
                               VAR_DOS_SEQ.Device.AVJ216.EnableCnd := FALSE;
                               VAR_DOS_SEQ.Device.AVJ217.AutoCnd := FALSE;                                             (* STEP: 73 Tank Hema Drain Valve*)
                               VAR_DOS_SEQ.Device.AVJ217.EnableCnd := FALSE;
                               VAR_DOS_SEQ.Device.AVJ218.AutoCnd := TRUE;                                              (* STEP: 73 Recirculation Valve*)
                               VAR_DOS_SEQ.Device.AVJ218.EnableCnd := FALSE;
                               VAR_DOS_SEQ.Device.AVJ221.AutoCnd := FALSE;                                             (* STEP: 73 Inlet Loop Valve*)
                               VAR_DOS_SEQ.Device.AVJ221.EnableCnd := FALSE;
                               VAR_DOS_SEQ.Device.AVJ230.AutoCnd := FALSE;                                              (* STEP: 73 *)
                               VAR_DOS_SEQ.Device.AVJ230.EnableCnd := FALSE;
                               VAR_DOS_SEQ.Device.AVJ231.AutoCnd := TRUE;                                              (* STEP: 73 *)
                               VAR_DOS_SEQ.Device.AVJ231.EnableCnd := FALSE;
                               VAR_DOS_SEQ.Device.AVJ232.AutoCnd := FALSE;                                             (* STEP: 73 *)
                               VAR_DOS_SEQ.Device.AVJ232.EnableCnd := FALSE;
                               VAR_DOS_SEQ.Device.AVJ233.AutoCnd := FALSE;                                             (* STEP: 73 *)
                               VAR_DOS_SEQ.Device.AVJ233.EnableCnd := FALSE;
                               VAR_DOS_SEQ.Device.AVJ234.AutoCnd := TRUE;                                              (* STEP: 73 *)
                               VAR_DOS_SEQ.Device.AVJ234.EnableCnd := FALSE;
                               VAR_DOS_SEQ.Device.AVJ235.AutoCnd := FALSE;                                             (* STEP: 73 *)
                               VAR_DOS_SEQ.Device.AVJ235.EnableCnd := FALSE;

                               VAR_DOS_SEQ.Device.LTJ203.ALR_HighLimitEn := TRUE;                                      (* STEP: 73 Hema Tank Level*)
                               VAR_DOS_SEQ.Device.LTJ203.ALR_HighLimitSP := HMI_PAM_3._607;
                               VAR_DOS_SEQ.Device.LTJ203.ALR_LowLimitEn := FALSE;
                               VAR_DOS_SEQ.Device.LTJ203.ALR_LowLimitSP := 0;
                               VAR_DOS_SEQ.Device.LTJ203.SP := HMI_PAM_3._626;
                               VAR_DOS_SEQ.Device.LTJ203.CMP := 2;
                               VAR_DOS_SEQ.Device.LTJ203.MinDev := 0;
                               VAR_DOS_SEQ.Device.LTJ203.MaxDev := 0;

                               VAR_DOS_SEQ.Device.TTJ203.ALR_HighLimitEn := TRUE;                                      (* STEP: 73 Hema Tank Temperature*)
                               VAR_DOS_SEQ.Device.TTJ203.ALR_HighLimitSP := HMI_PAM_3._620;
                               VAR_DOS_SEQ.Device.TTJ203.ALR_LowLimitEn := FALSE;
                               VAR_DOS_SEQ.Device.TTJ203.ALR_LowLimitSP := 0;
                               VAR_DOS_SEQ.Device.TTJ203.SP := HMI_PAM_3._633;
                               VAR_DOS_SEQ.Device.TTJ203.CMP := 2;
                               VAR_DOS_SEQ.Device.TTJ203.MinDev := 0;
                               VAR_DOS_SEQ.Device.TTJ203.MaxDev := 0;

                               VAR_DOS_SEQ.Device.LSJ200.ALR := FALSE;                                                 (* STEP: 73 *)
                               VAR_DOS_SEQ.Device.LSJ200.WAIT_OFF := FALSE;
                               VAR_DOS_SEQ.Device.LSJ200.WAIT_ON := FALSE;

                               VAR_DOS_SEQ.Device.LSJ201.ALR := FALSE;                                                 (* STEP: 73 *)
                               VAR_DOS_SEQ.Device.LSJ201.WAIT_OFF := FALSE;
                               VAR_DOS_SEQ.Device.LSJ201.WAIT_ON := FALSE;

                               VAR_DOS_SEQ.Device.LSJ202.ALR := FALSE;                                                 (* STEP: 73 *)
                               VAR_DOS_SEQ.Device.LSJ202.WAIT_OFF := FALSE;
                               VAR_DOS_SEQ.Device.LSJ202.WAIT_ON := FALSE;

                               VAR_DOS_SEQ.Device.FSJ201.ALR := FALSE;                                                 (* STEP: 73 *)
                               VAR_DOS_SEQ.Device.FSJ201.WAIT_OFF := FALSE;
                               VAR_DOS_SEQ.Device.FSJ201.WAIT_ON := FALSE;

                               VAR_DOS_SEQ.Device.FSJ202.ALR := FALSE;                                                 (* STEP: 73 *)
                               VAR_DOS_SEQ.Device.FSJ202.WAIT_OFF := FALSE;
                               VAR_DOS_SEQ.Device.FSJ202.WAIT_ON := FALSE;

                               VAR_DOS_SEQ.Mem.PBAbortEnable := TRUE;                                                  (* STEP: 73 PB Abort Sequence Enable*)
                               VAR_DOS_SEQ.Mem.PBStopEnable := TRUE;                                                   (* STEP: 73 PB Stop Sequence Enable*)
                               VAR_DOS_SEQ.Mem.PBStartEnable := FALSE;                                                 (* STEP: 73 PB Start Sequence Enable*)
                               VAR_DOS_SEQ.Mem.ContainersStop := TRUE;                                                 (* STEP: 73 *)
                               VAR_DOS_SEQ.Mem.MachineStart := TRUE;                                                   (* STEP: 73 *)
                               VAR_DOS_SEQ.Mem.MachineStop := FALSE;                                                   (* STEP: 73 *)
                               VAR_DOS_SEQ.Mem.DummyBottles := FALSE;                                                  (* STEP: 73 Dummy Bottle Install*)
                               VAR_DOS_SEQ.Mem.PositioningRequest := FALSE;                                            (* STEP: 73 Request of Cam Positioning at height SP of Sequncer*)
                               VAR_DOS_SEQ.Mem.COP_Cycle := FALSE;                                                     (* STEP: 73 COP Cycle Check Requested*)
                               VAR_DOS_SEQ.Mem.LapsCounter := FALSE;                                                   (* STEP: 73 *)
                               VAR_DOS_SEQ.Mem.ValveOpening := FALSE;                                                  (* STEP: 73 *)
                               VAR_DOS_SEQ.Mem.CopAfterCipRequest := FALSE;                                            (* STEP: 73 Request Of Cop After Cip*)

                               VAR_DOS_SEQ.ITC.CIP_CleaningRequest := TRUE;                                            (* STEP: 73 To CIP -> Request of Solution Sending*)
                               VAR_DOS_SEQ.ITC.CIP_Alarm := FALSE;                                                     (* STEP: 73 To CIP -> Critical Alarm Present*)
                               VAR_DOS_SEQ.ITC.CIP_RinseEnded := FALSE;                                                (* STEP: 73 To CIP -> Rinse Finished*)
                               VAR_DOS_SEQ.ITC.CIP_ChangeEnded := FALSE;                                               (* STEP: 73 To CIP -> Change Finished*)
                               VAR_DOS_SEQ.ITC.CIP_DrainRunning := FALSE;                                              (* STEP: 73 To CIP -> Drain Cycle Running*)
                               VAR_DOS_SEQ.ITC.CIP_RinseRunning := FALSE;                                              (* STEP: 73 To CIP -> Rinse Cycle Running*)
                               VAR_DOS_SEQ.ITC.CIP_CleaningRunning := TRUE;                                            (* STEP: 73 To CIP -> Cleaning Cycle Running*)
                               VAR_DOS_SEQ.ITC.CIP_DrainEnded := FALSE;                                                (* STEP: 73 To CIP -> Drain Finished*)
                               VAR_DOS_SEQ.ITC.CIP_FloodingEnded := FALSE;                                             (* STEP: 73 To CIP -> Flooding Finished*)
                               VAR_DOS_SEQ.ITC.CIP_FlipEnable := FALSE;                                                (* STEP: 73 *)
                               VAR_DOS_SEQ.ITC.CIP_CycleEnded := FALSE;                                                (* STEP: 73 *)

                               VAR_DOS_SEQ.ITC.PROD_ReadyForHeating := FALSE;                                          (* STEP: 73 To PASTO -> Filler Ready for Production (Heating)*)
                               VAR_DOS_SEQ.ITC.PROD_DoserInTemperature := FALSE;                                       (* STEP: 73 To PASTO -> Filler Temperature OK (After Heating)*)
                               VAR_DOS_SEQ.ITC.PROD_ProductRequest := FALSE;                                           (* STEP: 73 To PASTO -> Product Request*)
                               VAR_DOS_SEQ.ITC.PROD_DoserOnFillingMode := FALSE;                                       (* STEP: 73 To PASTO -> Product Consumend -Filling Valve Opening*)
                               VAR_DOS_SEQ.ITC.PROD_EndProductionCompleted := FALSE;                                   (* STEP: 73 To PASTO -> End Production Done*)
                               VAR_DOS_SEQ.ITC.PROD_ProductRecoveryEnd := FALSE;                                       (* STEP: 73 To PASTO -> Product Recovery End*)
                               VAR_DOS_SEQ.ITC.PROD_WaterRequestAfterProd := FALSE;                                    (* STEP: 73 To PASTO -> Water Request For Filler Rinse Afetr Production*)

                       74: (* Spare Steps *)

                       75: (* CIP - Piston washing *)

                               VAR_DOS_SEQ.Device.PPJ201_PID.PID_Enable := FALSE;                                      (* STEP: 75 Doser Recovery Pump*)
                               VAR_DOS_SEQ.Device.PPJ201_PID.PID_Mode := FALSE;
                               VAR_DOS_SEQ.Device.PPJ201_PID.Auto_SP_Value := 0;
                               VAR_DOS_SEQ.Device.PPJ201_PID.FIX_Value := 0;

                               VAR_DOS_SEQ.Device.PPJ202_PID.PID_Enable := TRUE;                                       (* STEP: 75 Doser Recovery Pump*)
                               VAR_DOS_SEQ.Device.PPJ202_PID.PID_Mode := FALSE;
                               VAR_DOS_SEQ.Device.PPJ202_PID.Auto_SP_Value := 0;
                               VAR_DOS_SEQ.Device.PPJ202_PID.FIX_Value := HMI_PAM_3._630;

                               VAR_DOS_SEQ.Device.PPJ203_PID.PID_Enable := FALSE;                                      (* STEP: 75 Diaphragm Pump for Recovery pulp*)
                               VAR_DOS_SEQ.Device.PPJ203_PID.PID_Mode := FALSE;
                               VAR_DOS_SEQ.Device.PPJ203_PID.Auto_SP_Value := 0;
                               VAR_DOS_SEQ.Device.PPJ203_PID.FIX_Value := 0;

                               VAR_DOS_SEQ.Device.MMJ201_PID.PID_Enable := TRUE;                                       (* STEP: 75 Shaker Motor*)
                               VAR_DOS_SEQ.Device.MMJ201_PID.PID_Mode := FALSE;
                               VAR_DOS_SEQ.Device.MMJ201_PID.Auto_SP_Value := 0;
                               VAR_DOS_SEQ.Device.MMJ201_PID.FIX_Value := 15;

                               VAR_DOS_SEQ.Device.RVJ201_PID.PID_Enable := FALSE;                                      (* STEP: 75 *)
                               VAR_DOS_SEQ.Device.RVJ201_PID.PID_Mode := FALSE;
                               VAR_DOS_SEQ.Device.RVJ201_PID.Auto_SP_Value := 0;
                               VAR_DOS_SEQ.Device.RVJ201_PID.FIX_Value := 0;

                               VAR_DOS_SEQ.Device.AVJ201.AutoCnd := FALSE;                                             (* STEP: 75 Inlet Valve*)
                               VAR_DOS_SEQ.Device.AVJ201.EnableCnd := FALSE;
                               VAR_DOS_SEQ.Device.AVJ210.AutoCnd := FALSE;                                             (* STEP: 75 Washing Duct Valve*)
                               VAR_DOS_SEQ.Device.AVJ210.EnableCnd := FALSE;
                               VAR_DOS_SEQ.Device.AVJ211.AutoCnd := TRUE;                                              (* STEP: 75 Sprayball Valve*)
                               VAR_DOS_SEQ.Device.AVJ211.EnableCnd := TRUE;
                               VAR_DOS_SEQ.Device.AVJ212.AutoCnd := TRUE;                                              (* STEP: 75 *)
                               VAR_DOS_SEQ.Device.AVJ212.EnableCnd := TRUE;
                               VAR_DOS_SEQ.Device.AVJ215.AutoCnd := FALSE;                                             (* STEP: 75 Atmospheric drain valve*)
                               VAR_DOS_SEQ.Device.AVJ215.EnableCnd := FALSE;
                               VAR_DOS_SEQ.Device.AVJ216.AutoCnd := TRUE;                                              (* STEP: 75 Recirculation Valve*)
                               VAR_DOS_SEQ.Device.AVJ216.EnableCnd := FALSE;
                               VAR_DOS_SEQ.Device.AVJ217.AutoCnd := TRUE;                                              (* STEP: 75 Tank Hema Drain Valve*)
                               VAR_DOS_SEQ.Device.AVJ217.EnableCnd := TRUE;
                               VAR_DOS_SEQ.Device.AVJ218.AutoCnd := TRUE;                                              (* STEP: 75 Recirculation Valve*)
                               VAR_DOS_SEQ.Device.AVJ218.EnableCnd := FALSE;
                               VAR_DOS_SEQ.Device.AVJ221.AutoCnd := FALSE;                                             (* STEP: 75 Inlet Loop Valve*)
                               VAR_DOS_SEQ.Device.AVJ221.EnableCnd := FALSE;
                               VAR_DOS_SEQ.Device.AVJ230.AutoCnd := TRUE;                                              (* STEP: 75 *)
                               VAR_DOS_SEQ.Device.AVJ230.EnableCnd := TRUE;
                               VAR_DOS_SEQ.Device.AVJ231.AutoCnd := TRUE;                                              (* STEP: 75 *)
                               VAR_DOS_SEQ.Device.AVJ231.EnableCnd := FALSE;
                               VAR_DOS_SEQ.Device.AVJ232.AutoCnd := FALSE;                                             (* STEP: 75 *)
                               VAR_DOS_SEQ.Device.AVJ232.EnableCnd := FALSE;
                               VAR_DOS_SEQ.Device.AVJ233.AutoCnd := TRUE;                                              (* STEP: 75 *)
                               VAR_DOS_SEQ.Device.AVJ233.EnableCnd := FALSE;
                               VAR_DOS_SEQ.Device.AVJ234.AutoCnd := TRUE;                                              (* STEP: 75 *)
                               VAR_DOS_SEQ.Device.AVJ234.EnableCnd := FALSE;
                               VAR_DOS_SEQ.Device.AVJ235.AutoCnd := FALSE;                                             (* STEP: 75 *)
                               VAR_DOS_SEQ.Device.AVJ235.EnableCnd := FALSE;

                               VAR_DOS_SEQ.Device.LTJ203.ALR_HighLimitEn := TRUE;                                      (* STEP: 75 Hema Tank Level*)
                               VAR_DOS_SEQ.Device.LTJ203.ALR_HighLimitSP := HMI_PAM_3._607;
                               VAR_DOS_SEQ.Device.LTJ203.ALR_LowLimitEn := TRUE;
                               VAR_DOS_SEQ.Device.LTJ203.ALR_LowLimitSP := HMI_PAM_3._606;
                               VAR_DOS_SEQ.Device.LTJ203.SP := HMI_PAM_3._626;
                               VAR_DOS_SEQ.Device.LTJ203.CMP := 2;
                               VAR_DOS_SEQ.Device.LTJ203.MinDev := 0;
                               VAR_DOS_SEQ.Device.LTJ203.MaxDev := 0;

                               VAR_DOS_SEQ.Device.TTJ203.ALR_HighLimitEn := TRUE;                                      (* STEP: 75 Hema Tank Temperature*)
                               VAR_DOS_SEQ.Device.TTJ203.ALR_HighLimitSP := HMI_PAM_3._620;
                               VAR_DOS_SEQ.Device.TTJ203.ALR_LowLimitEn := FALSE;
                               VAR_DOS_SEQ.Device.TTJ203.ALR_LowLimitSP := 0;
                               VAR_DOS_SEQ.Device.TTJ203.SP := HMI_PAM_3._633;
                               VAR_DOS_SEQ.Device.TTJ203.CMP := 2;
                               VAR_DOS_SEQ.Device.TTJ203.MinDev := 0;
                               VAR_DOS_SEQ.Device.TTJ203.MaxDev := 0;

                               VAR_DOS_SEQ.Device.LSJ200.ALR := FALSE;                                                 (* STEP: 75 *)
                               VAR_DOS_SEQ.Device.LSJ200.WAIT_OFF := FALSE;
                               VAR_DOS_SEQ.Device.LSJ200.WAIT_ON := FALSE;

                               VAR_DOS_SEQ.Device.LSJ201.ALR := FALSE;                                                 (* STEP: 75 *)
                               VAR_DOS_SEQ.Device.LSJ201.WAIT_OFF := FALSE;
                               VAR_DOS_SEQ.Device.LSJ201.WAIT_ON := FALSE;

                               VAR_DOS_SEQ.Device.LSJ202.ALR := FALSE;                                                 (* STEP: 75 *)
                               VAR_DOS_SEQ.Device.LSJ202.WAIT_OFF := FALSE;
                               VAR_DOS_SEQ.Device.LSJ202.WAIT_ON := FALSE;

                               VAR_DOS_SEQ.Device.FSJ201.ALR := FALSE;                                                 (* STEP: 75 *)
                               VAR_DOS_SEQ.Device.FSJ201.WAIT_OFF := FALSE;
                               VAR_DOS_SEQ.Device.FSJ201.WAIT_ON := FALSE;

                               VAR_DOS_SEQ.Device.FSJ202.ALR := FALSE;                                                 (* STEP: 75 *)
                               VAR_DOS_SEQ.Device.FSJ202.WAIT_OFF := FALSE;
                               VAR_DOS_SEQ.Device.FSJ202.WAIT_ON := FALSE;

                               VAR_DOS_SEQ.Mem.PBAbortEnable := TRUE;                                                  (* STEP: 75 PB Abort Sequence Enable*)
                               VAR_DOS_SEQ.Mem.PBStopEnable := TRUE;                                                   (* STEP: 75 PB Stop Sequence Enable*)
                               VAR_DOS_SEQ.Mem.PBStartEnable := FALSE;                                                 (* STEP: 75 PB Start Sequence Enable*)
                               VAR_DOS_SEQ.Mem.ContainersStop := TRUE;                                                 (* STEP: 75 *)
                               VAR_DOS_SEQ.Mem.MachineStart := TRUE;                                                   (* STEP: 75 *)
                               VAR_DOS_SEQ.Mem.MachineStop := FALSE;                                                   (* STEP: 75 *)
                               VAR_DOS_SEQ.Mem.DummyBottles := FALSE;                                                  (* STEP: 75 Dummy Bottle Install*)
                               VAR_DOS_SEQ.Mem.PositioningRequest := FALSE;                                            (* STEP: 75 Request of Cam Positioning at height SP of Sequncer*)
                               VAR_DOS_SEQ.Mem.COP_Cycle := FALSE;                                                     (* STEP: 75 COP Cycle Check Requested*)
                               VAR_DOS_SEQ.Mem.LapsCounter := FALSE;                                                   (* STEP: 75 *)
                               VAR_DOS_SEQ.Mem.ValveOpening := FALSE;                                                  (* STEP: 75 *)
                               VAR_DOS_SEQ.Mem.CopAfterCipRequest := FALSE;                                            (* STEP: 75 Request Of Cop After Cip*)

                               VAR_DOS_SEQ.ITC.CIP_CleaningRequest := TRUE;                                            (* STEP: 75 To CIP -> Request of Solution Sending*)
                               VAR_DOS_SEQ.ITC.CIP_Alarm := FALSE;                                                     (* STEP: 75 To CIP -> Critical Alarm Present*)
                               VAR_DOS_SEQ.ITC.CIP_RinseEnded := FALSE;                                                (* STEP: 75 To CIP -> Rinse Finished*)
                               VAR_DOS_SEQ.ITC.CIP_ChangeEnded := FALSE;                                               (* STEP: 75 To CIP -> Change Finished*)
                               VAR_DOS_SEQ.ITC.CIP_DrainRunning := FALSE;                                              (* STEP: 75 To CIP -> Drain Cycle Running*)
                               VAR_DOS_SEQ.ITC.CIP_RinseRunning := FALSE;                                              (* STEP: 75 To CIP -> Rinse Cycle Running*)
                               VAR_DOS_SEQ.ITC.CIP_CleaningRunning := TRUE;                                            (* STEP: 75 To CIP -> Cleaning Cycle Running*)
                               VAR_DOS_SEQ.ITC.CIP_DrainEnded := FALSE;                                                (* STEP: 75 To CIP -> Drain Finished*)
                               VAR_DOS_SEQ.ITC.CIP_FloodingEnded := TRUE;                                              (* STEP: 75 To CIP -> Flooding Finished*)
                               VAR_DOS_SEQ.ITC.CIP_FlipEnable := FALSE;                                                (* STEP: 75 *)
                               VAR_DOS_SEQ.ITC.CIP_CycleEnded := FALSE;                                                (* STEP: 75 *)

                               VAR_DOS_SEQ.ITC.PROD_ReadyForHeating := FALSE;                                          (* STEP: 75 To PASTO -> Filler Ready for Production (Heating)*)
                               VAR_DOS_SEQ.ITC.PROD_DoserInTemperature := FALSE;                                       (* STEP: 75 To PASTO -> Filler Temperature OK (After Heating)*)
                               VAR_DOS_SEQ.ITC.PROD_ProductRequest := FALSE;                                           (* STEP: 75 To PASTO -> Product Request*)
                               VAR_DOS_SEQ.ITC.PROD_DoserOnFillingMode := FALSE;                                       (* STEP: 75 To PASTO -> Product Consumend -Filling Valve Opening*)
                               VAR_DOS_SEQ.ITC.PROD_EndProductionCompleted := FALSE;                                   (* STEP: 75 To PASTO -> End Production Done*)
                               VAR_DOS_SEQ.ITC.PROD_ProductRecoveryEnd := FALSE;                                       (* STEP: 75 To PASTO -> Product Recovery End*)
                               VAR_DOS_SEQ.ITC.PROD_WaterRequestAfterProd := FALSE;                                    (* STEP: 75 To PASTO -> Water Request For Filler Rinse Afetr Production*)

                       76: (* Spare Steps *)

                       77: (* CIP - Filling valve washing *)

                               VAR_DOS_SEQ.Device.PPJ201_PID.PID_Enable := FALSE;                                      (* STEP: 77 Doser Recovery Pump*)
                               VAR_DOS_SEQ.Device.PPJ201_PID.PID_Mode := FALSE;
                               VAR_DOS_SEQ.Device.PPJ201_PID.Auto_SP_Value := 0;
                               VAR_DOS_SEQ.Device.PPJ201_PID.FIX_Value := 0;

                               VAR_DOS_SEQ.Device.PPJ202_PID.PID_Enable := TRUE;                                       (* STEP: 77 Doser Recovery Pump*)
                               VAR_DOS_SEQ.Device.PPJ202_PID.PID_Mode := FALSE;
                               VAR_DOS_SEQ.Device.PPJ202_PID.Auto_SP_Value := 0;
                               VAR_DOS_SEQ.Device.PPJ202_PID.FIX_Value := HMI_PAM_3._630;

                               VAR_DOS_SEQ.Device.PPJ203_PID.PID_Enable := FALSE;                                      (* STEP: 77 Diaphragm Pump for Recovery pulp*)
                               VAR_DOS_SEQ.Device.PPJ203_PID.PID_Mode := FALSE;
                               VAR_DOS_SEQ.Device.PPJ203_PID.Auto_SP_Value := 0;
                               VAR_DOS_SEQ.Device.PPJ203_PID.FIX_Value := 0;

                               VAR_DOS_SEQ.Device.MMJ201_PID.PID_Enable := TRUE;                                       (* STEP: 77 Shaker Motor*)
                               VAR_DOS_SEQ.Device.MMJ201_PID.PID_Mode := FALSE;
                               VAR_DOS_SEQ.Device.MMJ201_PID.Auto_SP_Value := 0;
                               VAR_DOS_SEQ.Device.MMJ201_PID.FIX_Value := 15;

                               VAR_DOS_SEQ.Device.RVJ201_PID.PID_Enable := FALSE;                                      (* STEP: 77 *)
                               VAR_DOS_SEQ.Device.RVJ201_PID.PID_Mode := FALSE;
                               VAR_DOS_SEQ.Device.RVJ201_PID.Auto_SP_Value := 0;
                               VAR_DOS_SEQ.Device.RVJ201_PID.FIX_Value := 0;

                               VAR_DOS_SEQ.Device.AVJ201.AutoCnd := FALSE;                                             (* STEP: 77 Inlet Valve*)
                               VAR_DOS_SEQ.Device.AVJ201.EnableCnd := FALSE;
                               VAR_DOS_SEQ.Device.AVJ210.AutoCnd := FALSE;                                             (* STEP: 77 Washing Duct Valve*)
                               VAR_DOS_SEQ.Device.AVJ210.EnableCnd := FALSE;
                               VAR_DOS_SEQ.Device.AVJ211.AutoCnd := TRUE;                                              (* STEP: 77 Sprayball Valve*)
                               VAR_DOS_SEQ.Device.AVJ211.EnableCnd := TRUE;
                               VAR_DOS_SEQ.Device.AVJ212.AutoCnd := TRUE;                                              (* STEP: 77 *)
                               VAR_DOS_SEQ.Device.AVJ212.EnableCnd := TRUE;
                               VAR_DOS_SEQ.Device.AVJ215.AutoCnd := FALSE;                                             (* STEP: 77 Atmospheric drain valve*)
                               VAR_DOS_SEQ.Device.AVJ215.EnableCnd := FALSE;
                               VAR_DOS_SEQ.Device.AVJ216.AutoCnd := TRUE;                                              (* STEP: 77 Recirculation Valve*)
                               VAR_DOS_SEQ.Device.AVJ216.EnableCnd := FALSE;
                               VAR_DOS_SEQ.Device.AVJ217.AutoCnd := TRUE;                                              (* STEP: 77 Tank Hema Drain Valve*)
                               VAR_DOS_SEQ.Device.AVJ217.EnableCnd := TRUE;
                               VAR_DOS_SEQ.Device.AVJ218.AutoCnd := TRUE;                                              (* STEP: 77 Recirculation Valve*)
                               VAR_DOS_SEQ.Device.AVJ218.EnableCnd := FALSE;
                               VAR_DOS_SEQ.Device.AVJ221.AutoCnd := FALSE;                                             (* STEP: 77 Inlet Loop Valve*)
                               VAR_DOS_SEQ.Device.AVJ221.EnableCnd := FALSE;
                               VAR_DOS_SEQ.Device.AVJ230.AutoCnd := TRUE;                                              (* STEP: 77 *)
                               VAR_DOS_SEQ.Device.AVJ230.EnableCnd := TRUE;
                               VAR_DOS_SEQ.Device.AVJ231.AutoCnd := TRUE;                                              (* STEP: 77 *)
                               VAR_DOS_SEQ.Device.AVJ231.EnableCnd := FALSE;
                               VAR_DOS_SEQ.Device.AVJ232.AutoCnd := FALSE;                                             (* STEP: 77 *)
                               VAR_DOS_SEQ.Device.AVJ232.EnableCnd := FALSE;
                               VAR_DOS_SEQ.Device.AVJ233.AutoCnd := TRUE;                                              (* STEP: 77 *)
                               VAR_DOS_SEQ.Device.AVJ233.EnableCnd := FALSE;
                               VAR_DOS_SEQ.Device.AVJ234.AutoCnd := TRUE;                                              (* STEP: 77 *)
                               VAR_DOS_SEQ.Device.AVJ234.EnableCnd := FALSE;
                               VAR_DOS_SEQ.Device.AVJ235.AutoCnd := FALSE;                                             (* STEP: 77 *)
                               VAR_DOS_SEQ.Device.AVJ235.EnableCnd := FALSE;

                               VAR_DOS_SEQ.Device.LTJ203.ALR_HighLimitEn := TRUE;                                      (* STEP: 77 Hema Tank Level*)
                               VAR_DOS_SEQ.Device.LTJ203.ALR_HighLimitSP := HMI_PAM_3._607;
                               VAR_DOS_SEQ.Device.LTJ203.ALR_LowLimitEn := TRUE;
                               VAR_DOS_SEQ.Device.LTJ203.ALR_LowLimitSP := HMI_PAM_3._606;
                               VAR_DOS_SEQ.Device.LTJ203.SP := HMI_PAM_3._626;
                               VAR_DOS_SEQ.Device.LTJ203.CMP := 2;
                               VAR_DOS_SEQ.Device.LTJ203.MinDev := 0;
                               VAR_DOS_SEQ.Device.LTJ203.MaxDev := 0;

                               VAR_DOS_SEQ.Device.TTJ203.ALR_HighLimitEn := TRUE;                                      (* STEP: 77 Hema Tank Temperature*)
                               VAR_DOS_SEQ.Device.TTJ203.ALR_HighLimitSP := HMI_PAM_3._620;
                               VAR_DOS_SEQ.Device.TTJ203.ALR_LowLimitEn := FALSE;
                               VAR_DOS_SEQ.Device.TTJ203.ALR_LowLimitSP := 0;
                               VAR_DOS_SEQ.Device.TTJ203.SP := HMI_PAM_3._633;
                               VAR_DOS_SEQ.Device.TTJ203.CMP := 2;
                               VAR_DOS_SEQ.Device.TTJ203.MinDev := 0;
                               VAR_DOS_SEQ.Device.TTJ203.MaxDev := 0;

                               VAR_DOS_SEQ.Device.LSJ200.ALR := FALSE;                                                 (* STEP: 77 *)
                               VAR_DOS_SEQ.Device.LSJ200.WAIT_OFF := FALSE;
                               VAR_DOS_SEQ.Device.LSJ200.WAIT_ON := FALSE;

                               VAR_DOS_SEQ.Device.LSJ201.ALR := FALSE;                                                 (* STEP: 77 *)
                               VAR_DOS_SEQ.Device.LSJ201.WAIT_OFF := FALSE;
                               VAR_DOS_SEQ.Device.LSJ201.WAIT_ON := FALSE;

                               VAR_DOS_SEQ.Device.LSJ202.ALR := FALSE;                                                 (* STEP: 77 *)
                               VAR_DOS_SEQ.Device.LSJ202.WAIT_OFF := FALSE;
                               VAR_DOS_SEQ.Device.LSJ202.WAIT_ON := FALSE;

                               VAR_DOS_SEQ.Device.FSJ201.ALR := FALSE;                                                 (* STEP: 77 *)
                               VAR_DOS_SEQ.Device.FSJ201.WAIT_OFF := FALSE;
                               VAR_DOS_SEQ.Device.FSJ201.WAIT_ON := FALSE;

                               VAR_DOS_SEQ.Device.FSJ202.ALR := FALSE;                                                 (* STEP: 77 *)
                               VAR_DOS_SEQ.Device.FSJ202.WAIT_OFF := FALSE;
                               VAR_DOS_SEQ.Device.FSJ202.WAIT_ON := FALSE;

                               VAR_DOS_SEQ.Mem.PBAbortEnable := TRUE;                                                  (* STEP: 77 PB Abort Sequence Enable*)
                               VAR_DOS_SEQ.Mem.PBStopEnable := TRUE;                                                   (* STEP: 77 PB Stop Sequence Enable*)
                               VAR_DOS_SEQ.Mem.PBStartEnable := FALSE;                                                 (* STEP: 77 PB Start Sequence Enable*)
                               VAR_DOS_SEQ.Mem.ContainersStop := TRUE;                                                 (* STEP: 77 *)
                               VAR_DOS_SEQ.Mem.MachineStart := TRUE;                                                   (* STEP: 77 *)
                               VAR_DOS_SEQ.Mem.MachineStop := FALSE;                                                   (* STEP: 77 *)
                               VAR_DOS_SEQ.Mem.DummyBottles := FALSE;                                                  (* STEP: 77 Dummy Bottle Install*)
                               VAR_DOS_SEQ.Mem.PositioningRequest := FALSE;                                            (* STEP: 77 Request of Cam Positioning at height SP of Sequncer*)
                               VAR_DOS_SEQ.Mem.COP_Cycle := FALSE;                                                     (* STEP: 77 COP Cycle Check Requested*)
                               VAR_DOS_SEQ.Mem.LapsCounter := FALSE;                                                   (* STEP: 77 *)
                               VAR_DOS_SEQ.Mem.ValveOpening := TRUE;                                                   (* STEP: 77 *)
                               VAR_DOS_SEQ.Mem.CopAfterCipRequest := FALSE;                                            (* STEP: 77 Request Of Cop After Cip*)

                               VAR_DOS_SEQ.ITC.CIP_CleaningRequest := TRUE;                                            (* STEP: 77 To CIP -> Request of Solution Sending*)
                               VAR_DOS_SEQ.ITC.CIP_Alarm := FALSE;                                                     (* STEP: 77 To CIP -> Critical Alarm Present*)
                               VAR_DOS_SEQ.ITC.CIP_RinseEnded := FALSE;                                                (* STEP: 77 To CIP -> Rinse Finished*)
                               VAR_DOS_SEQ.ITC.CIP_ChangeEnded := FALSE;                                               (* STEP: 77 To CIP -> Change Finished*)
                               VAR_DOS_SEQ.ITC.CIP_DrainRunning := FALSE;                                              (* STEP: 77 To CIP -> Drain Cycle Running*)
                               VAR_DOS_SEQ.ITC.CIP_RinseRunning := FALSE;                                              (* STEP: 77 To CIP -> Rinse Cycle Running*)
                               VAR_DOS_SEQ.ITC.CIP_CleaningRunning := TRUE;                                            (* STEP: 77 To CIP -> Cleaning Cycle Running*)
                               VAR_DOS_SEQ.ITC.CIP_DrainEnded := FALSE;                                                (* STEP: 77 To CIP -> Drain Finished*)
                               VAR_DOS_SEQ.ITC.CIP_FloodingEnded := FALSE;                                             (* STEP: 77 To CIP -> Flooding Finished*)
                               VAR_DOS_SEQ.ITC.CIP_FlipEnable := FALSE;                                                (* STEP: 77 *)
                               VAR_DOS_SEQ.ITC.CIP_CycleEnded := FALSE;                                                (* STEP: 77 *)
```
